PROGRAM PRG_NC_ReadWriteParameters
VAR

	ReadWriteParameters			: FB_NC_ReadWriteParameters;

END_VAR


ReadWriteParameters.Cmd_ReadParameters;
ReadWriteParameters.Cmd_WriteParameters;
ReadWriteParameters.Set_EncoderDemoninator;
ReadWriteParameters.Set_EncoderNuminator;
ReadWriteParameters.Set_EncoderOffset;
ReadWriteParameters.Set_ModuloValue;

ReadWriteParameters(
	Cmd_ReadParameters:= , 
	Cmd_WriteParameters:= , 
	Set_EncoderNuminator:= , 
	Set_EncoderDemoninator:= , 
	Set_EncoderOffset:= , 
	Set_ModuloValue:= , 
	Sts_MaximumVelocity=> , 
	Sts_MaximumAcceleration=> , 
	Sts_Maximumdeceleration=> , 
	Sts_EncoderNuminator=> , 
	Sts_EncoderDemoninator=> , 
	Sts_EncoderOffset=> , 
	Sts_ModuloValue=> , 
	Sts_StatusSTRING=> , 
	Axis:=Main.Axis01 );

END_PROGRAM

(* stored: Version 1.1.0.1, ProductVersion 3.1.4024.14
   POU PRG_NC_ReadWriteParameters: Id {d5db72a3-cf91-4f33-ba58-a951fc505340}, SpecialFunc None *)
